//==================================================================================================
//							Beckhoff Automation Poland
//									06.02.2024
//	Basic Axis Function Block object to control mostly used functionabilities, 
//	Required libs: Tc2_EtherCAT, Tc2_MC2_Drive, Tc2_MC2
// 	v2.0	|| TC v 3.1.4024.53		|| New release. Inheritance added.
//  v1.6	|| TC v 3.1.4024.22		|| Added structure ST_MotionPowerData. Reading parameters inside it.
//  v1.5	|| TC v 3.1.4022.27		|| Added error description (string type)
// 	v1.4 	|| TC v 3.1.4022.20	 	|| ACT_MotorMonitoring - only for real axis
// 	v1.3 	|| TC v 3.1.4022.16	 	|| Common interface similar to AX5000
// 	v1.2 	|| TC v 3.1.4022.16	 	|| Added ACT_SetPositionIO, migration part of logic from ACT_SetPosition to ACT_SetPositionIO
// 	v1.1 	|| TC v 3.1.4022.16	 	|| ACT_MotorMonitoring - is executing always, ACT_Initialization - optimalization
// 	v1.0 	|| TC v 3.1.4022.16	 	|| First release
//==================================================================================================
{attribute 'reflection'}
FUNCTION_BLOCK FB_McAxisOnline_AX8xxx EXTENDS FB_McAxisOnline_NC
VAR_INPUT
END_VAR
VAR_OUTPUT
END_VAR
VAR
	fbSetPositionOffset					: FB_CoEAX8000SetPositionOffset;
	fbMotorMonitoring					: FB_MotorMonitoringAX8000;
	fbHoldingBrakeCtrl					: FB_HoldingBrakeCtrlAX8000;
	tonGetDriveDiag						: TON;
	fbReadChannelErrorCode				: FB_ReadChannelErrorCodeAX8000;
	mcReadDriveAddress					: MC_ReadDriveAddress;
	fbGetDriveRef						: FB_GetDriveRef;
	
	bDriveAddressReady					: BOOL;
	bDriveRefReady						: BOOL;
END_VAR

// Device dependent initialization 
M_Init_AX8xxx();

// Device independent commands, mostly NC 
M_States();
M_SWLimitSwitch();
M_Stop();
M_Power();
M_Homing();
M_Jog();
M_Move();
M_Reset();
M_SetPosition();
// Device dependent commands
// Motor monitoring possible only with real axis
IF NOT AxisRef.Status.OpMode.SimulationAxis THEN
	M_MotorMonitoring();
END_IF
// Device dependent commands, possible only on real axis after complete initialization
IF bInitialized AND NOT AxisRef.Status.OpMode.SimulationAxis THEN
	M_SetPositionIO();
	M_DriveDiag();
	M_HoldingBrakeCtrl();
END_IF

// Device independent error collection
M_ErrorCollection();

METHOD M_DriveDiag : BOOL
VAR_INPUT
END_VAR
// Auto update when drive error
tonGetDriveDiag(IN:= Axis.stError.bDriveError AND NOT tonGetDriveDiag.Q, PT:= T#5S, Q=> , ET=> );

fbReadChannelErrorCode(	bExecute				:= Axis.stChannelErrorCode.bExecute OR tonGetDriveDiag.Q,
						stDriveRef				:= Axis.stDriveRef,
						bBusy					=> Axis.stChannelErrorCode.bBusy,
						bError					=> Axis.stChannelErrorCode.bError,
						iAdsErrId				=> Axis.stChannelErrorCode.uiAdsErrId,
						iCANopenErrId			=> Axis.stChannelErrorCode.uiSecErrId,
						uiChannelErrorCode		=> Axis.stChannelErrorCode.uiChannelErrorCode,
						uiChannelErrorCodeHex	=> Axis.stChannelErrorCode.uiChannelErrorCodeHex);
END_METHOD

METHOD M_ErrorCollection : BOOL
VAR_INPUT
END_VAR
// Error flags
Axis.stError.bDriveError					:= AxisRef.Status.DriveDeviceError;

Axis.stError.bNcError						:= AxisRef.Status.Error;

Axis.stError.bFBError						:= Axis.mcPower.bError OR Axis.mcReset.bError OR Axis.mcHome.bError OR Axis.mcJog.bError
													OR Axis.mcHalt.bError OR Axis.mcStop.bError OR Axis.mcSS1.bError OR Axis.mcSS2.bError
													OR Axis.mcMoveAbsolute.bError OR Axis.mcMoveRelative.bError OR Axis.mcMoveVelocity.bError OR Axis.mcMoveModulo.bError
													OR Axis.mcMoveAbsolute2.bError OR Axis.mcMoveRelative2.bError OR Axis.mcMoveVelocity2.bError OR Axis.mcMoveModulo2.bError
													OR Axis.stNcLimitSwitch.bError OR Axis.mcSetPosition.bError;
									
Axis.stError.bCommunicationError			:= Axis.stChannelErrorCode.bError OR Axis.stSetPositionOffset.bError OR Axis.stMotorMonitoring.bError OR Axis.stHoldingBrake.bError;

Axis.stError.bError							:= Axis.stError.bDriveError OR Axis.stError.bNcError OR Axis.stError.bFBError OR Axis.stError.bCommunicationError;
Axis.bError									:= Axis.stError.bError; // Forward one stage up

// Error codes
Axis.stError.uiDriveErrorID 				:= Axis.stChannelErrorCode.uiChannelErrorCode;
Axis.stError.uiDriveErrorIDHex 				:= Axis.stChannelErrorCode.uiChannelErrorCodeHex;

Axis.stError.udiNcErrorID 					:= AxisRef.Status.ErrorID;
Axis.stError.udiNcErrorIDHex 				:= AxisRef.Status.ErrorID;
	

Axis.stError.udiFBErrorID 					:= 	Axis.mcPower.udiErrorID + 
												Axis.mcReset.udiErrorID + 
												Axis.mcHome.udiErrorID + 
												Axis.mcJog.udiErrorID +
												Axis.mcHalt.udiErrorID + 
												Axis.mcStop.udiErrorID + 
												Axis.mcSS1.udiErrorID + 
												Axis.mcSS2.udiErrorID +
												Axis.mcMoveAbsolute.udiErrorID + 
												Axis.mcMoveRelative.udiErrorID + 
												Axis.mcMoveVelocity.udiErrorID + 
												Axis.mcMoveModulo.udiErrorID +
												Axis.mcMoveAbsolute2.udiErrorID + 
												Axis.mcMoveRelative2.udiErrorID + 
												Axis.mcMoveVelocity2.udiErrorID + 
												Axis.mcMoveModulo2.udiErrorID +
												Axis.stNcLimitSwitch.udiErrorID + 
												Axis.mcSetPosition.udiErrorID;

Axis.stError.udiFBErrorIDHex 				:= Axis.stError.udiFBErrorID;

Axis.stError.udiErrorID						:= Axis.stSetPositionOffset.udiErrorID;
Axis.stError.uiAdsErrorID					:= Axis.stChannelErrorCode.uiAdsErrId + Axis.stMotorMonitoring.uiAdsErrId + Axis.stHoldingBrake.uiAdsErrId;
Axis.stError.uiSecErrorID					:= Axis.stChannelErrorCode.uiSecErrId + Axis.stMotorMonitoring.uiSecErrId + Axis.stHoldingBrake.uiSecErrId;

Axis.stError.sNcError						:= F_AxErrMsg(Axis.stError.udiNcErrorID);
Axis.stError.sDriveError					:= F_AX8xErrMsg(Axis.stError.uiDriveErrorID);
END_METHOD

METHOD M_HoldingBrakeCtrl : BOOL
VAR_INPUT
END_VAR
fbHoldingBrakeCtrl(	bForceLock			:= Axis.stHoldingBrake.bForceLock,
					bForceUnlock		:= Axis.stHoldingBrake.bForceUnlock,
					stDriveRef			:= Axis.stDriveRef,
					bBusy				=> Axis.stHoldingBrake.bBusy,
					bError				=> Axis.stHoldingBrake.bError,
					iAdsErrId			=> Axis.stHoldingBrake.uiAdsErrId,
					iCANopenErrId		=> Axis.stHoldingBrake.uiSecErrId);
END_METHOD

METHOD M_Init_AX8xxx : BOOL
VAR_INPUT
END_VAR
// bInitialized flag is set just once. 
// bReInitialized ise set each time we do online change or request reinit operation
// bDriveAddressReady, bReadParameterSetReady, bDriveRefReady - set just once after successed read

// Online change detection
bOnlineChangeDetected					:= udiOnlineChangeCntOld <> TwinCAT_SystemInfoVarList._AppInfo.OnlineChangeCnt;
udiOnlineChangeCntOld 					:= TwinCAT_SystemInfoVarList._AppInfo.OnlineChangeCnt;
// Reset init
IF bReInit OR bOnlineChangeDetected THEN
	iInitStep							:= 0;
END_IF

//Initialization process
CASE iInitStep OF
	0:	// Read Drive Address
		
		Axis.mcReadDriveAddress.bExecute	:=	 TRUE;
		iInitStep						:= iInitStep + 10;
		
	10: // Wait for data
	
		IF NOT Axis.mcReadDriveAddress.bBusy THEN
			Axis.mcReadDriveAddress.bExecute	:=	 FALSE;
			IF Axis.mcReadDriveAddress.bDone THEN
				iInitStep 				:= iInitStep + 10;
				bDriveAddressReady 		:= TRUE;
			ELSE
				iInitStep 				:= 1000;		// Error step
			END_IF
		END_IF
		
	20:	// Read Parameter Set
		
		Axis.mcReadParameterSet.bExecute		:=	 TRUE;
		iInitStep						:= iInitStep + 10;
		
	30: // Wait for data
	
		IF NOT Axis.mcReadParameterSet.bBusy THEN
			Axis.mcReadParameterSet.bExecute	:=	 FALSE;
			IF Axis.mcReadParameterSet.bDone THEN
				iInitStep 				:= iInitStep + 10;
				bReadParameterSetReady 	:= TRUE;
			ELSE
				iInitStep 				:= 1000;		// Error step
			END_IF
		END_IF	
	
	40:	// Get Drive Ref
		
		Axis.stGetDriveRef.bExecute		:=	 TRUE;
		iInitStep						:= iInitStep + 10;
		
	50: // Wait for data
	
		IF NOT Axis.stGetDriveRef.bBusy THEN
			Axis.stGetDriveRef.bExecute	:=	 FALSE;
			IF NOT Axis.stGetDriveRef.bError THEN
				iInitStep 				:= iInitStep + 10;
				bDriveRefReady 			:= TRUE;
			ELSE
				iInitStep 				:= 1000;		// Error step
			END_IF
		END_IF
	
	60: // Success - initialized flag, clear error
		bReInitialized					:= bInitialized;	// TRUE only when it's not first initialization e.g. online change
		bInitialized 					:= TRUE;
		bReInitializationError			:= FALSE;			// TRUE only when it's not first initialization e.g. online change
		bInitializationError			:= FALSE;
		iInitStep 						:= iInitStep + 10;
		
	70: // Idle
	
		;
		
	1000: // Error step
		wInitializationErrorCounter 	:= wInitializationErrorCounter + 1;
		IF wInitializationErrorCounter < 100 THEN
			iInitStep					:= iInitStep + 5;			// Go to delay
		ELSE
			bReInitializationError		:= bInitializationError;	// TRUE only when it's not first initialization e.g. online change
			bInitializationError		:= TRUE;
			bReInitialized				:= FALSE;
			iInitStep 					:= iInitStep + 10;
		END_IF

	1005: // Delay step
		tonDelay(IN:= TRUE, PT:= T#1S);
		IF tonDelay.Q THEN
			tonDelay(IN:= FALSE, PT:= T#1S);
			iInitStep					:= 0;
		END_IF
		
	1010: // Idle after error
		;
	
END_CASE

mcReadDriveAddress(	Axis				:= AxisRef,
					Execute				:= Axis.mcReadDriveAddress.bExecute,
					Done				=> Axis.mcReadDriveAddress.bDone,
					Busy				=> Axis.mcReadDriveAddress.bBusy,
					Error				=> Axis.mcReadDriveAddress.bError,
					ErrorID				=> Axis.mcReadDriveAddress.udiErrorID,
					DriveAddress		=> Axis.stDriveAddress);
				
mcReadParameterSet(	Parameter			:= Axis.stAxisParameter,
					Axis				:= AxisRef,
					Execute				:= Axis.mcReadParameterSet.bExecute,
					Done				=> Axis.mcReadParameterSet.bDone,
					Busy				=> Axis.mcReadParameterSet.bBusy,
					Error				=> Axis.mcReadParameterSet.bError,
					ErrorID				=> Axis.mcReadParameterSet.udiErrorID);
					
fbGetDriveRef(		bExecute			:= Axis.stGetDriveRef.bExecute,
					bBusy				=> Axis.stGetDriveRef.bBusy,
					bError				=> Axis.stGetDriveRef.bError,
					udiErrorID			=> Axis.stGetDriveRef.udiErrorID,
					stDriveRef			=> Axis.stDriveRef,
					Axis				:= AxisRef);
END_METHOD

METHOD M_MotorMonitoring : BOOL
VAR_INPUT
END_VAR
fbMotorMonitoring(	bReset				:= Axis.stMotorMonitoring.bReset,
					rTorqueLimit		:= Axis.stMotorMonitoring.rTorqueLimit,
					stDriveRef			:= Axis.stDriveRef,
					bError				=> Axis.stMotorMonitoring.bError,
					uiAdsErrId			=> Axis.stMotorMonitoring.uiAdsErrId,
					uiCANopenErrId		=> Axis.stMotorMonitoring.uiSecErrId,
					bInitialized		=> Axis.stMotorMonitoring.bInitialized,
					bWarning			=> Axis.stMotorMonitoring.bWarning,
					rWarningCurrent		=> Axis.stMotorMonitoring.rWarningCurrent,
					rTorquePerc			=> Axis.stMotorMonitoring.rTorquePerc,
					rTorquePercMax		=> Axis.stMotorMonitoring.rTorquePercMax,
					rTorque				=> Axis.stMotorMonitoring.rTorque,
					rTorqueF			=> Axis.stMotorMonitoring.rTorqueF,
					rTorqueMax			=> Axis.stMotorMonitoring.rTorqueMax,
					rCurrent			=> Axis.stMotorMonitoring.rCurrent,
					rCurrentF			=> Axis.stMotorMonitoring.rCurrentF,
					rCurrentMax			=> Axis.stMotorMonitoring.rCurrentMax,
					rI2T				=> Axis.stMotorMonitoring.rI2T,
					rI2TMax				=> Axis.stMotorMonitoring.rI2TMax,
					stPowerData			=> Axis.stMotorMonitoring.stPowerData,
					Axis				:= AxisRef);
END_METHOD

METHOD M_SetPositionIO : BOOL
VAR_INPUT
END_VAR
fbSetPositionOffset(Execute				:= Axis.stSetPositionOffset.bExecute,
					Position			:= Axis.stSetPositionOffset.lrPosition,
					Relative			:= Axis.stSetPositionOffset.bRelative,
					Feedback			:= Axis.stSetPositionOffset.eFeedback,
					Memory				:= Axis.stSetPositionOffset.eMemory,
					Busy				=> Axis.stSetPositionOffset.bBusy,
					Error				=> Axis.stSetPositionOffset.bError,
					ErrorID				=> Axis.stSetPositionOffset.udiErrorID,
					Axis				:= AxisRef);
END_METHOD

END_FUNCTION_BLOCK

(* stored: Version 1.1.0.1, ProductVersion 3.1.4024.15
   POU FB_McAxisOnline_AX8xxx: Id {9f989287-2df8-4d7a-9dbf-e015c53994f2}, SpecialFunc None
   Method M_DriveDiag: Id {84a965f3-e766-48c7-b448-9dd0db8d9919}
   Method M_ErrorCollection: Id {e02898c0-ab01-41eb-a9c6-6238aaeab901}
   Method M_HoldingBrakeCtrl: Id {7eb9470b-52c1-410c-a31b-9195f72a347b}
   Method M_Init_AX8xxx: Id {7b8b56bc-c154-49ad-becc-f212291f4184}
   Method M_MotorMonitoring: Id {22af2b36-cbee-4162-b094-47ccb6f6de63}
   Method M_SetPositionIO: Id {648cd4b1-b42f-4317-8f58-1250bb2256d7} *)
